Fanuc KAREL source: kd00011.KL

-- PROVISIONAL review KL for V770-1; original PC SHA256 bf0bcfd9d8374267626bc603c94b71a0d4402f721ab99fb5e5b3296f9b07f549
-- Incomplete behavior may be omitted. Consult companion uncertainty JSON. Do not deploy.
PROGRAM KD00011
%NOLOCKGROUP
VAR
  I : INTEGER
  J : INTEGER
  B : BOOLEAN
  R : REAL
  S : STRING[80]
BEGIN
  -- UNRESOLVED_PC offsets 5-6; opcodes 15
  -- UNRESOLVED_PC offsets 11-15; opcodes 7F
END KD00011
